FUNCTION_BLOCK PLC_RW_M262 (* Composite Function Block Type *)
  (* Standard: 61499-2 *)
  (* Version 0.0, 6/30/2025, azam_w, Schneider Electric, template *)
  PACKAGE Main;
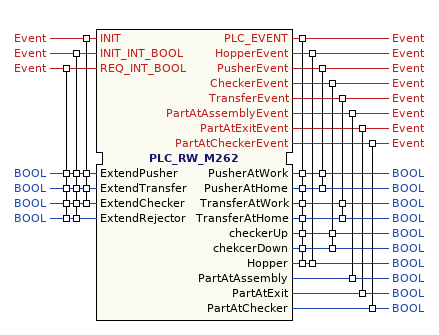
  EVENT_INPUT
    INIT WITH ExtendTransfer, ExtendChecker, ExtendPusher;
    INIT_INT_BOOL WITH ExtendPusher, ExtendTransfer, ExtendChecker, ExtendRejector;
    REQ_INT_BOOL WITH ExtendPusher, ExtendTransfer, ExtendChecker, ExtendRejector;
  END_EVENT
  EVENT_OUTPUT
    PLC_EVENT WITH PusherAtWork, PusherAtHome, TransferAtWork, TransferAtHome, checkerUp, chekcerDown, Hopper;
    HopperEvent WITH Hopper;
    PusherEvent WITH PusherAtWork, PusherAtHome;
    CheckerEvent WITH checkerUp, chekcerDown;
    TransferEvent WITH TransferAtWork, TransferAtHome;
    PartAtAssemblyEvent WITH PartAtAssembly;
    PartAtExitEvent WITH PartAtExit;
    PartAtCheckerEvent WITH PartAtChecker;
  END_EVENT
  VAR_INPUT
    ExtendPusher : BOOL;
    ExtendTransfer : BOOL;
    ExtendChecker : BOOL;
    ExtendRejector : BOOL;
  END_VAR
  VAR_OUTPUT
    PusherAtWork : BOOL;
    PusherAtHome : BOOL;
    TransferAtWork : BOOL;
    TransferAtHome : BOOL;
    checkerUp : BOOL;
    chekcerDown : BOOL;
    Hopper : BOOL;
    PartAtAssembly : BOOL;
    PartAtExit : BOOL;
    PartAtChecker : BOOL;
  END_VAR
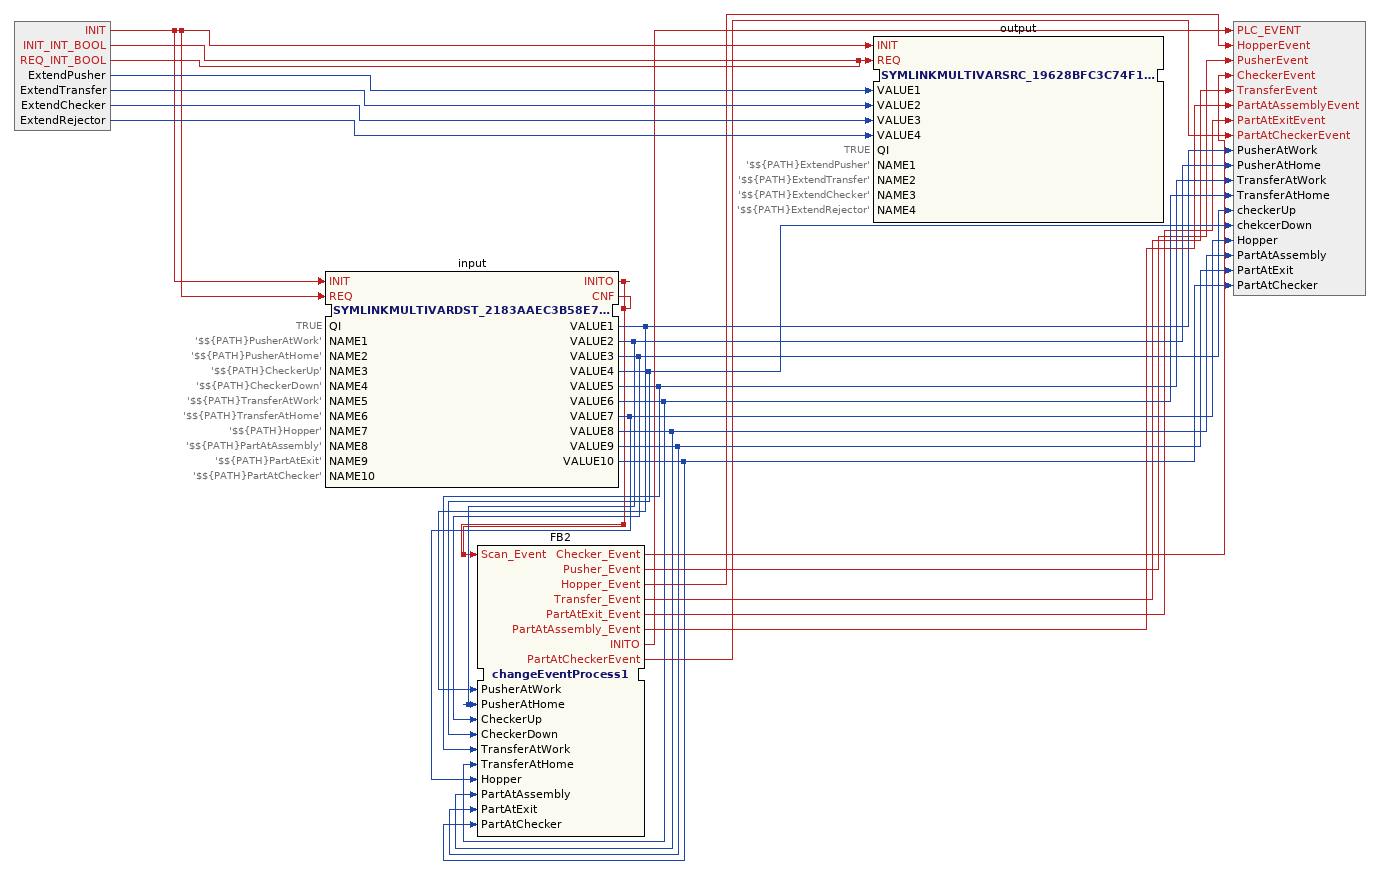
  FBS
    input : SYMLINKMULTIVARDST_2183AAEC3B58E76C9(QI := TRUE, NAME1 := '$${PATH}PusherAtWork', NAME2 := '$${PATH}PusherAtHome', NAME3 := '$${PATH}CheckerUp', NAME4 := '$${PATH}CheckerDown', NAME5 := '$${PATH}TransferAtWork', NAME6 := '$${PATH}TransferAtHome', NAME7 := '$${PATH}Hopper', NAME8 := '$${PATH}PartAtAssembly', NAME9 := '$${PATH}PartAtExit', NAME10 := '$${PATH}PartAtChecker'); {SET_ATTRIBUTE(Configuration.GenericFBType.InterfaceParams, Runtime.System#I:=10;VALUE${I$}:BOOL,BOOL,BOOL,BOOL,BOOL,BOOL,BOOL,BOOL,BOOL,BOOL)}
    output : SYMLINKMULTIVARSRC_19628BFC3C74F1AB1(QI := TRUE, NAME1 := '$${PATH}ExtendPusher', NAME2 := '$${PATH}ExtendTransfer', NAME3 := '$${PATH}ExtendChecker', NAME4 := '$${PATH}ExtendRejector'); {SET_ATTRIBUTE(Configuration.GenericFBType.InterfaceParams, Runtime.System#I:=4;VALUE${I$}:BOOL,BOOL,BOOL,BOOL)}
    FB2 : changeEventProcess1;
  END_FBS
  EVENT_CONNECTIONS
    FB2.Checker_Event TO CheckerEvent;
    FB2.Pusher_Event TO PusherEvent;
    FB2.Hopper_Event TO HopperEvent;
    FB2.Transfer_Event TO TransferEvent;
    FB2.PartAtExit_Event TO PartAtExitEvent;
    FB2.PartAtAssembly_Event TO PartAtAssemblyEvent;
    FB2.INITO TO PLC_EVENT;
    INIT TO input.INIT;
    INIT TO input.REQ;
    input.INITO TO FB2.Scan_Event;
    input.CNF TO FB2.Scan_Event;
    FB2.PartAtCheckerEvent TO PartAtCheckerEvent;
    INIT TO output.INIT;
    INIT_INT_BOOL TO output.REQ;
    REQ_INT_BOOL TO output.REQ;
  END_CONNECTIONS
  DATA_CONNECTIONS
    input.VALUE1 TO PusherAtWork;
    input.VALUE1 TO FB2.PusherAtWork;
    input.VALUE2 TO PusherAtHome;
    input.VALUE2 TO FB2.PusherAtHome;
    input.VALUE3 TO checkerUp;
    input.VALUE3 TO FB2.CheckerUp;
    input.VALUE4 TO chekcerDown;
    input.VALUE4 TO FB2.CheckerDown;
    input.VALUE5 TO TransferAtWork;
    input.VALUE5 TO FB2.TransferAtWork;
    input.VALUE6 TO TransferAtHome;
    input.VALUE6 TO FB2.TransferAtHome;
    input.VALUE7 TO Hopper;
    input.VALUE7 TO FB2.Hopper;
    input.VALUE8 TO PartAtAssembly;
    input.VALUE8 TO FB2.PartAtAssembly;
    input.VALUE9 TO PartAtExit;
    input.VALUE9 TO FB2.PartAtExit;
    input.VALUE10 TO PartAtChecker;
    input.VALUE10 TO FB2.PartAtChecker;
    ExtendPusher TO output.VALUE1;
    ExtendTransfer TO output.VALUE2;
    ExtendChecker TO output.VALUE3;
    ExtendRejector TO output.VALUE4;
  END_CONNECTIONS
END_FUNCTION_BLOCK
